FUNCTION F_DecIndex : INT
VAR_INPUT
	IDX:	INT;		// Index to be incremented
	IdxMIN:	INT;		// Min Value for index	
	IdxMAX:	INT;		// Max Value for index
END_VAR
VAR
END_VAR

IF IDX > IdxMIN THEN
	F_DecIndex := IDX - 1; 
ELSIF IDX = IdxMIN THEN
	F_DecIndex := IdxMAX;
ELSIF IDX < IdxMIN OR IDX > IdxMAX THEN
	F_DecIndex := IdxMAX;
END_IF

END_FUNCTION

(* stored: Version 1.1.0.1, ProductVersion 3.1.4024.4
   POU F_DecIndex: Id {42ed4245-7b0e-420c-b8af-51eb070817ff}, SpecialFunc None *)
